FUNCTION Celcius_to_Fahrenet : REAL
VAR_INPUT
	fCelcius: REAL;
	
END_VAR
VAR
END_VAR

Celcius_to_Fahrenet := fCelcius * 1.8 +32.0 ;

END_FUNCTION

(* stored: Version 1.1.0.1, ProductVersion 3.1.4024.9
   POU Celcius_to_Fahrenet: Id {1721cd38-099d-4b26-b004-a0780ea9c5d7}, SpecialFunc None *)
